TYPE typeSettings :
	STRUCT
		TextName:STRING := ('Unnamed Setting');
		Value:INT;
	END_STRUCT
END_TYPE

(* stored: Version 1.1.0.1, ProductVersion 3.1.4024.11
   DUT typeSettings: Id {e14b704a-4d02-0678-389a-2c87526d053b} *)
